{attribute 'GeneratedUsingTerminal: EL1258-0010-0017'}
{attribute addProperty BoxType "EL1258-0010-0017"}
{attribute addProperty Id "MTI_Inputs_1x_Channel_1AT %I*MTI_Inputs_1x_Channel_CC1B212F11MTI_Inputs_1x_Channel_2AT %I*MTI_Inputs_1x_Channel_CC1B212F11MTI_Inputs_1x_Channel_3AT %I*MTI_Inputs_1x_Channel_CC1B212F11MTI_Inputs_1x_Channel_4AT %I*MTI_Inputs_1x_Channel_CC1B212F11MTI_Inputs_1x_Channel_5AT %I*MTI_Inputs_1x_Channel_CC1B212F11MTI_Inputs_1x_Channel_6AT %I*MTI_Inputs_1x_Channel_CC1B212F11MTI_Inputs_1x_Channel_7AT %I*MTI_Inputs_1x_Channel_CC1B212F11MTI_Inputs_1x_Channel_8AT %I*MTI_Inputs_1x_Channel_CC1B212F11MTI_Outputs_Channel_1AT %Q*MTI_Outputs_Channel_0F1028A12MTI_Outputs_Channel_2AT %Q*MTI_Outputs_Channel_0F1028A12MTI_Outputs_Channel_3AT %Q*MTI_Outputs_Channel_0F1028A12MTI_Outputs_Channel_4AT %Q*MTI_Outputs_Channel_0F1028A12MTI_Outputs_Channel_5AT %Q*MTI_Outputs_Channel_0F1028A12MTI_Outputs_Channel_6AT %Q*MTI_Outputs_Channel_0F1028A12MTI_Outputs_Channel_7AT %Q*MTI_Outputs_Channel_0F1028A12MTI_Outputs_Channel_8AT %Q*MTI_Outputs_Channel_0F1028A12WcStateAT %I*WcState_9091E0EB2InfoDataAT %I*InfoData_BEF6B88E18"}
{attribute addProperty CRC "1771991042"}
{attribute addProperty Size "124"}
TYPE EL1258_699E7002 :
STRUCT
	{attribute addProperty Name "MTI_Inputs_1x_Channel_1"}
	MTI_Inputs_1x_Channel_1 : MTI_Inputs_1x_Channel_CC1B212F;
	{attribute addProperty Name "MTI_Inputs_1x_Channel_2"}
	MTI_Inputs_1x_Channel_2 : MTI_Inputs_1x_Channel_CC1B212F;
	{attribute addProperty Name "MTI_Inputs_1x_Channel_3"}
	MTI_Inputs_1x_Channel_3 : MTI_Inputs_1x_Channel_CC1B212F;
	{attribute addProperty Name "MTI_Inputs_1x_Channel_4"}
	MTI_Inputs_1x_Channel_4 : MTI_Inputs_1x_Channel_CC1B212F;
	{attribute addProperty Name "MTI_Inputs_1x_Channel_5"}
	MTI_Inputs_1x_Channel_5 : MTI_Inputs_1x_Channel_CC1B212F;
	{attribute addProperty Name "MTI_Inputs_1x_Channel_6"}
	MTI_Inputs_1x_Channel_6 : MTI_Inputs_1x_Channel_CC1B212F;
	{attribute addProperty Name "MTI_Inputs_1x_Channel_7"}
	MTI_Inputs_1x_Channel_7 : MTI_Inputs_1x_Channel_CC1B212F;
	{attribute addProperty Name "MTI_Inputs_1x_Channel_8"}
	MTI_Inputs_1x_Channel_8 : MTI_Inputs_1x_Channel_CC1B212F;
	{attribute addProperty Name "MTI_Outputs_Channel_1"}
	MTI_Outputs_Channel_1 : MTI_Outputs_Channel_0F1028A1;
	{attribute addProperty Name "MTI_Outputs_Channel_2"}
	MTI_Outputs_Channel_2 : MTI_Outputs_Channel_0F1028A1;
	{attribute addProperty Name "MTI_Outputs_Channel_3"}
	MTI_Outputs_Channel_3 : MTI_Outputs_Channel_0F1028A1;
	{attribute addProperty Name "MTI_Outputs_Channel_4"}
	MTI_Outputs_Channel_4 : MTI_Outputs_Channel_0F1028A1;
	{attribute addProperty Name "MTI_Outputs_Channel_5"}
	MTI_Outputs_Channel_5 : MTI_Outputs_Channel_0F1028A1;
	{attribute addProperty Name "MTI_Outputs_Channel_6"}
	MTI_Outputs_Channel_6 : MTI_Outputs_Channel_0F1028A1;
	{attribute addProperty Name "MTI_Outputs_Channel_7"}
	MTI_Outputs_Channel_7 : MTI_Outputs_Channel_0F1028A1;
	{attribute addProperty Name "MTI_Outputs_Channel_8"}
	MTI_Outputs_Channel_8 : MTI_Outputs_Channel_0F1028A1;
	{attribute addProperty Name "WcState"}
	WcState : WcState_9091E0EB;
	{attribute addProperty Name "InfoData"}
	InfoData : InfoData_BEF6B88E;
END_STRUCT
END_TYPE

(* stored: Version 1.2.0.0, ProductVersion 3.1.4024.9
   DUT EL1258_699E7002: Id {4f3c4c33-c1ba-4395-a5b7-a5ae5229b656} *)
